Omron Sysmac Studio project tcp_ip_nx1p2_solution_thanh (Sysmac Studio 1.45.1.64010, StandardProject)

# Controller new_Controller_0: NX1P2-9024DT version 1.40
Task PrimaryTask (priority 4, period or condition 2000): Program0
Library MTCP_Server_NJNX 2.6. (contents left out)
Library OEN_Communication_V1_0_22 1.0.22 (contents left out)

PROGRAM Program0
VAR
    Tcp_Send : BOOL;
    tcp_connect : SktTCPConnect;
    Dest_adrress_ip : STRING[256];
    dest_adress_port : UINT;
    tcp_connect_done : BOOL;
    tcp_clear_buf : SktClearBuf;
    Socket_Dummy : _sSOCKET;
    tcp_clear_buf_done : BOOL;
    tcp_get_status : SktGetTCPStatus;
    tcp_get_status_done : BOOL;
    tcp_send_data : SktTCPSend;
    Data_send : ARRAY[0..5] OF BYTE;
    DATA_RECEI : ARRAY[0..5] OF BYTE;
    TCP_SEND_DONE : BOOL;
    TCP_RECEI_DATA : SktTCPRcv;
    TCP_RECEI_DONE : BOOL;
    TCP_CLOSE_CONNECTION : SktClose;
    RESET_TPC_CLIENT : RS;
    TCP_LISTEN : BOOL;
    TCPSERVER_CLOSE_DONE : BOOL;
    TCP_ACCEPT_DONE : BOOL;
    TCP_SERVER_ACCPEPT : SktTCPAccept;
    SERVER_DATA_RECEI : ARRAY[0..4] OF BYTE;
    SERVER_DATA_SEND : ARRAY[0..4] OF BYTE;
    TCP_SERVER_RECEI_DATA : SktTCPRcv;
    TPC_SERVER_RECEI_DONE : BOOL;
    TCP_SERVER_RECEI_DONE : BOOL;
    TCP_SERVER_SEND_DONE : BOOL;
    TCP_SERVER_SEND : SktTCPSend;
    TCP_SERVER_CLOSE : SktClose;
    TCP_LIBRARY_OPEN : BOOL;
    MODBUSTCP_REGISTER : ARRAY[0..25] OF WORD;
    MODBUSACCESS_LIST : ARRAY[0..5] OF OEN\Modbus\sModbusAccess;
    MODBUS_COIL : ARRAY[0..5] OF BOOL;
    MODBUS_INPUT : ARRAY[0..10] OF BOOL;
    MODBUS_INPUT_REGISTER : ARRAY[0..10] OF WORD;
    MODBUS_HOLDING_REGISTER : ARRAY[0..10] OF WORD;
    FB_MODBUS_TCP_LIBRARY : OEN\Modbus\ModbusTCP_Server;
END_VAR

(* Section tcp_client: ladder, written here as Structured Text *)

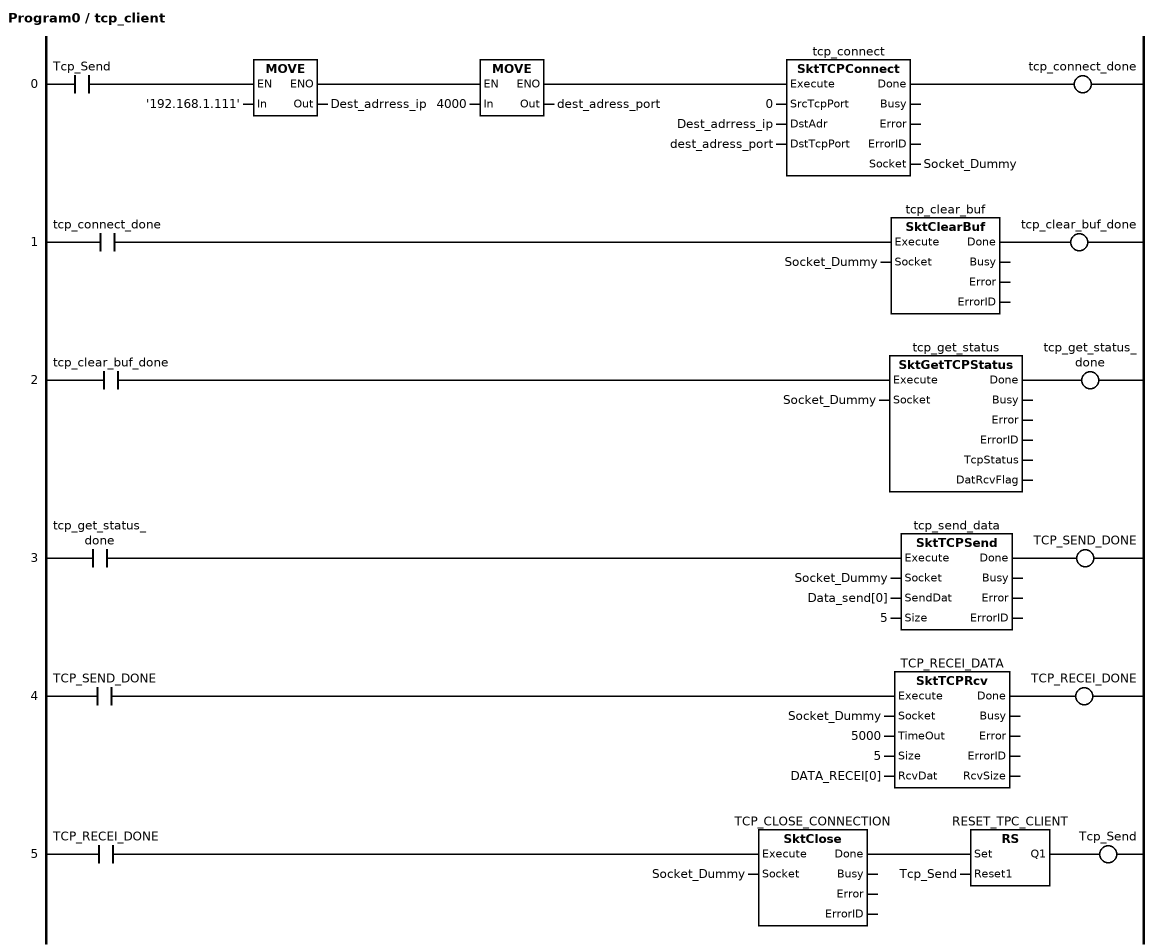
(* Rung 0 *)
IF Tcp_Send THEN
    Dest_adrress_ip := '192.168.1.111';
    dest_adress_port := 4000;
END_IF;
tcp_connect(Execute := Tcp_Send, SrcTcpPort := 0, DstAdr := Dest_adrress_ip, DstTcpPort := dest_adress_port, Socket => Socket_Dummy);
tcp_connect_done := tcp_connect.Done;
(* Rung 1 *)
tcp_clear_buf(Execute := tcp_connect_done, Socket := Socket_Dummy);
tcp_clear_buf_done := tcp_clear_buf.Done;
(* Rung 2 *)
tcp_get_status(Execute := tcp_clear_buf_done, Socket := Socket_Dummy);
tcp_get_status_done := tcp_get_status.Done;
(* Rung 3 *)
tcp_send_data(Execute := tcp_get_status_done, Socket := Socket_Dummy, SendDat := Data_send[0], Size := 5);
TCP_SEND_DONE := tcp_send_data.Done;
(* Rung 4 *)
TCP_RECEI_DATA(Execute := TCP_SEND_DONE, Socket := Socket_Dummy, TimeOut := 5000, Size := 5, RcvDat := DATA_RECEI[0]);
TCP_RECEI_DONE := TCP_RECEI_DATA.Done;
(* Rung 5 *)
TCP_CLOSE_CONNECTION(Execute := TCP_RECEI_DONE, Socket := Socket_Dummy);
RESET_TPC_CLIENT(Set := TCP_CLOSE_CONNECTION.Done, Reset1 := Tcp_Send);
Tcp_Send := RESET_TPC_CLIENT.Q1;

(* Section TCP_SERVER: ladder, written here as Structured Text *)

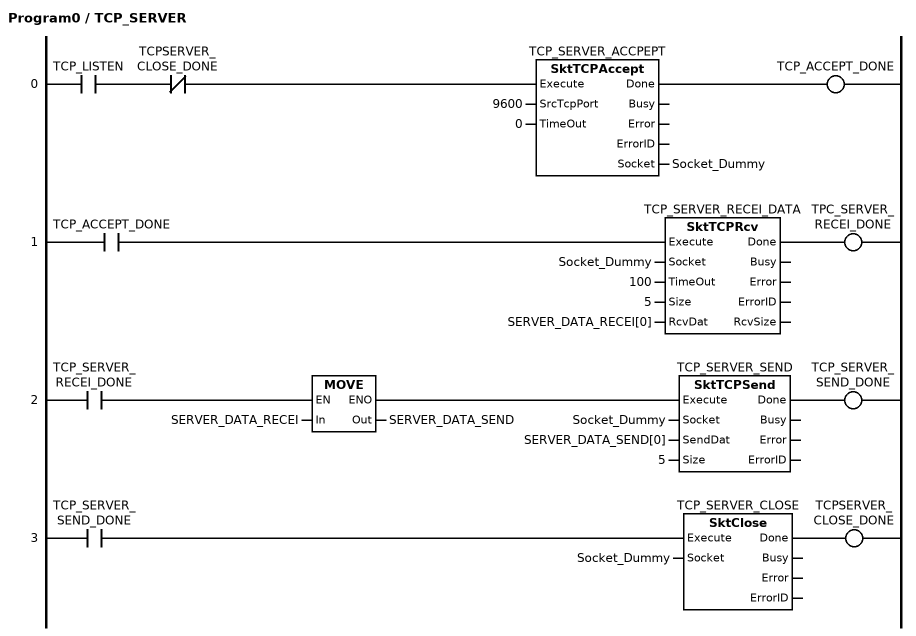
(* Rung 0 *)
TCP_SERVER_ACCPEPT(Execute := TCP_LISTEN AND NOT TCPSERVER_CLOSE_DONE, SrcTcpPort := 9600, TimeOut := 0, Socket => Socket_Dummy);
TCP_ACCEPT_DONE := TCP_SERVER_ACCPEPT.Done;
(* Rung 1 *)
TCP_SERVER_RECEI_DATA(Execute := TCP_ACCEPT_DONE, Socket := Socket_Dummy, TimeOut := 100, Size := 5, RcvDat := SERVER_DATA_RECEI[0]);
TPC_SERVER_RECEI_DONE := TCP_SERVER_RECEI_DATA.Done;
(* Rung 2 *)
IF TCP_SERVER_RECEI_DONE THEN SERVER_DATA_SEND := SERVER_DATA_RECEI; END_IF;
TCP_SERVER_SEND(Execute := TCP_SERVER_RECEI_DONE, Socket := Socket_Dummy, SendDat := SERVER_DATA_SEND[0], Size := 5);
TCP_SERVER_SEND_DONE := TCP_SERVER_SEND.Done;
(* Rung 3 *)
TCP_SERVER_CLOSE(Execute := TCP_SERVER_SEND_DONE, Socket := Socket_Dummy);
TCPSERVER_CLOSE_DONE := TCP_SERVER_CLOSE.Done;

(* Section tcp_server_library: ladder, written here as Structured Text *)

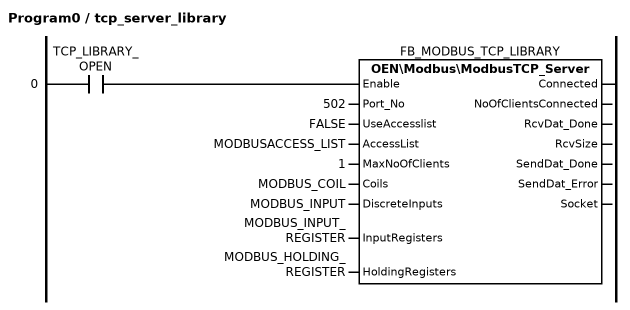
(* Rung 0 *)
FB_MODBUS_TCP_LIBRARY(Enable := TCP_LIBRARY_OPEN, Port_No := 502, UseAccesslist := FALSE, AccessList := MODBUSACCESS_LIST, MaxNoOfClients := 1, Coils := MODBUS_COIL, DiscreteInputs := MODBUS_INPUT, InputRegisters := MODBUS_INPUT_REGISTER, HoldingRegisters := MODBUS_HOLDING_REGISTER);
END_PROGRAM